// TIA Portal V18 export
TYPE "DT_FML_STATUS"
// stored: IsFailsafeCompliant false
   STRUCT
      Err : Bool;
      Cat : Int;
      ID : DInt;
   END_STRUCT;
END_TYPE
